TYPE stSubTank :
STRUCT
	//R//						
		error_code			:INT;
		state				:INT;
		Error				:BOOL;
	//W//
		Setoff				:BOOL;	//  
		timeout             :LREAL;//S
END_STRUCT
END_TYPE

(* stored: Version 1.1.0.1, ProductVersion 3.1.4024.11
   DUT stSubTank: Id {e9a53490-228b-497e-bd29-d25e8903f83a} *)
